TYPE AxesMuUnits :
(
	ARCSECONDS_PER_YEAR := 0,
	MILLIARCSECONDS_PER_YEAR := 1,
	DEGREES_PER_YEAR := 2,
	RADIANS_PER_YEAR := 3
);
END_TYPE

(* stored: Version 1.1.0.1, ProductVersion 3.1.4019.2
   DUT AxesMuUnits: Id {a56fa8c0-26d8-4705-bc13-d6fff6df6883} *)
